# EPICS substitutions: db/ecmcEL7332.substitutions
# All fields related to velocity scaling and alarms
file ecmcEL7332-chX.template
{
  pattern {CHAN,  LINR,    ESLO,   EOFF,   EGU,        PREC, LOW, LOLO, HIGH, HIHI, HYST, LLSV,       LSV,        HSV,        HHSV      }
          {0      "SLOPE", 1,      0,      "Raw",      0,    0,   0,    0,    0,    0,    "NO_ALARM", "NO_ALARM", "NO_ALARM", "NO_ALARM"}
          {1      "SLOPE", 1,      0,      "Raw",      0,    0,   0,    0,    0,    0,    "NO_ALARM", "NO_ALARM", "NO_ALARM", "NO_ALARM"}
}
